//Use this FB if NC-Reference mode is set to "Software Sync" or "Hardware-Sync".
//It is mandatory that the NC encoder parameter "Encoder Sub Mask (absolute range maximum value)" is set to the correct value!
//
//This FB checks the disctance between the falling edge of an reference sensor 
//and the final reference flag of the encoder (e.g. SingleTurn overflow in mode SoftwareSync)
//In case these two signals are very close together, it might be possible that the reference position varied about one motor turn
//depending whether the falling edge of the reference sensor occured before or after the software sync impulse.
//
//The FB reports an OK if the resulting distance if greater or equel than the "MinDistanceInDeg". 
{attribute 'no_check'}
FUNCTION_BLOCK AxSoftSyncDistance EXTENDS FbBase
VAR_OUTPUT CONSTANT
//option settings 
END_VAR
VAR CONSTANT
	DEG_PER_TURN											:	LREAL := 360.0;	
END_VAR
VAR_INPUT
	MinDistanceInDeg										:	LREAL := 45.0; //Minmum required distance between falling edge of sensor and software sync reference impuls (Single turn overflow)   
END_VAR
VAR_IN_OUT
	Axis													:	AXIS_REF;
END_VAR
VAR_OUTPUT
	Distance												: LREAL; //In user units (e.g. mm)
	DistancePerTurn											: LREAL; //In user units (e.g. mm)
	DistanceInDeg											: LREAL; //Resulting distance in degrees	
	OK														: BOOL;  //Inidcates whether the distance between falling edge of sensor and software sync is greater or equal than MinDistanceInDeg  
END_VAR
VAR
(*  Memory *****************************************************)
	LastErrorState											:	INT;
	LastErrorId												:	UDINT;
	ScalingNumerator										:	LREAL;
	ScalingDenumerator										:	LREAL;
	Scaling													:	LREAL;
	RefSystem												:	UDINT;
	RefMode													:	UDINT;
	{attribute 'displaymode':='hex'}
	EncSubMask												:	UDINT;


(*  Timer ******************************************************)

(*  Trigger ****************************************************)

(*  Blocks *****************************************************)
	ReadAdsPara												: ADSREAD := (NetID:= '' , Port:=AMSPORT_R0_NC,TmOut := DEFAULT_ADS_TIMEOUT );

(*  Error ******************************************************)
(*  Dummys *****************************************************)
	{attribute 'hide' := ''}
END_VAR

	(* Check distance between falling edge of reference sensor and deteced sync impulse		*)
	(****************************************************************************************)
	
(* Sequence ********************************************************)
	rtExecute(CLK := Execute);
	CASE state OF
	0 : 
		Busy 												:= FALSE;
		IF NOT Execute THEN
			OK												:= FALSE;
			Done 											:= FALSE;
			Error 											:= FALSE;
			ErrorID 										:= 0;
		END_IF
		IF rtExecute.Q THEN
			ReadAdsPara( Read := FALSE); 
			Busy											:= TRUE;
			Distance										:= 0.0;
			ScalingNumerator								:= 0.0;
			ScalingDenumerator								:= 0.0;
			Scaling											:= 0.0;
			RefSystem										:= 0;
			EncSubMask										:= 0;
			OK												:= FALSE;
			Done 											:= FALSE;
			Error 											:= FALSE;
			ErrorID 										:= 0;
			state 											:= state + 1;
		END_IF
		
		
	(* Read scaling numerator **********************************************)
	1:
		ReadAdsPara(Read:= TRUE,	IDxGrp:=(16#5000+Axis.NcToPlc.AxisId) , IDxOffs:=16#23,LEN:=SIZEOF(ScalingNumerator), DestAddr:=ADR(ScalingNumerator));	
		IF NOT ReadAdsPara.BUSY
		THEN
			IF ReadAdsPara.ERR
			THEN
				Busy										:= FALSE;
				Error										:= TRUE;
				ErrorID										:= ReadAdsPara.ERRID;
				LastErrorState								:= state;
				LastErrorId									:= ErrorId;
				state										:= 0;
			ELSE 
				state										:= state + 1;						
			END_IF
			ReadAdsPara( Read := FALSE);
		END_IF
		
	(* Read scaling denumerator **********************************************)
	2:
		ReadAdsPara(Read:= TRUE,	IDxGrp:=(16#5000+Axis.NcToPlc.AxisId) , IDxOffs:=16#24,LEN:=SIZEOF(ScalingDenumerator), DestAddr:=ADR(ScalingDenumerator));	
		IF NOT ReadAdsPara.BUSY
		THEN
			IF ReadAdsPara.ERR
			THEN
				Busy										:= FALSE;
				Error										:= TRUE;
				ErrorID										:= ReadAdsPara.ERRID;
				LastErrorState									:= state;
				LastErrorId									:= ErrorId;
				state										:= 0;
			ELSE
				Scaling										:= ScalingNumerator / SEL(ScalingDenumerator = 0.0, ScalingDenumerator , 1.0);	
				IF Scaling = 0.0
				THEN
					Busy									:= FALSE;
					Error									:= TRUE;
					ErrorID									:= MC_ERROR_PARAMETER_NOT_CORRECT;
					LastErrorState								:= state;
					LastErrorId									:= ErrorId;
					state									:= 0;	
				ELSE
					state									:= state + 1;
				END_IF					
			END_IF
			ReadAdsPara( Read := FALSE);
		END_IF

	(* Read distance in user units **********************************************)
	3:
		ReadAdsPara(Read:= TRUE,	IDxGrp:=(16#5100+Axis.NcToPlc.AxisId) , IDxOffs:=16#101,LEN:=SIZEOF(Distance), DestAddr:=ADR(Distance));	
		IF NOT ReadAdsPara.BUSY
		THEN
			IF ReadAdsPara.ERR
			THEN
				Busy										:= FALSE;
				Error										:= TRUE;
				ErrorID										:= ReadAdsPara.ERRID;
				LastErrorState									:= state;
				LastErrorId									:= ErrorId;
				state										:= 0;
			ELSE 
				state										:= state + 1;			
			END_IF
			ReadAdsPara( Read := FALSE);
		END_IF
		
	(* Read selected reference system **********************************************)
	4:
		ReadAdsPara(Read:= TRUE,	IDxGrp:=(16#5000+Axis.NcToPlc.AxisId) , IDxOffs:=16#19,LEN:=SIZEOF(RefSystem), DestAddr:=ADR(RefSystem));	
		IF NOT ReadAdsPara.BUSY
		THEN
			IF ReadAdsPara.ERR
			THEN
				Busy										:= FALSE;
				Error										:= TRUE;
				ErrorID										:= ReadAdsPara.ERRID;
				LastErrorState									:= state;
				LastErrorId									:= ErrorId;
				state										:= 0;
			ELSE 
				state										:= state + 1;					
			END_IF
			ReadAdsPara( Read := FALSE);
		END_IF
	
	(* Read selected reference mode **********************************************)
	5:
		ReadAdsPara(Read:= TRUE,	IDxGrp:=(16#5000+Axis.NcToPlc.AxisId) , IDxOffs:=16#107,LEN:=SIZEOF(RefMode), DestAddr:=ADR(RefMode));	
		IF NOT ReadAdsPara.BUSY
		THEN
			IF ReadAdsPara.ERR
			THEN
				Busy										:= FALSE;
				Error										:= TRUE;
				ErrorID										:= ReadAdsPara.ERRID;
				LastErrorState									:= state;
				LastErrorId									:= ErrorId;
				state										:= 0;
			ELSE 
				state										:= state + 1;					
			END_IF
			ReadAdsPara( Read := FALSE);
		END_IF
	
	(* Read EncSubMask (Inc per turn) **********************************************)
	6:
		ReadAdsPara(Read:= TRUE,	IDxGrp:=(16#5000+Axis.NcToPlc.AxisId) , IDxOffs:=16#108,LEN:=SIZEOF(EncSubMask), DestAddr:=ADR(EncSubMask));	
		IF NOT ReadAdsPara.BUSY
		THEN
			IF ReadAdsPara.ERR
			THEN
				Busy										:= FALSE;
				Error										:= TRUE;
				ErrorID										:= ReadAdsPara.ERRID;
				LastErrorState									:= state;
				LastErrorId									:= ErrorId;
				state										:= 0;
			ELSIF EncSubMask = 0
			THEN
				Busy										:= FALSE;
				Error										:= TRUE;
				ErrorID										:= MC_ERROR_PARAMETER_NOT_CORRECT;
				LastErrorState									:= state;
				LastErrorId									:= ErrorId;
				state										:= 0;			
			ELSE
				state										:= state + 1;					
			END_IF
			ReadAdsPara( Read := FALSE);
		END_IF
		
	(* Check reference value ************************************)
	7:
		DistancePerTurn										:= EncSubMask * Scaling;
		DistanceInDeg										:= (DEG_PER_TURN / DistancePerTurn) * Distance;	
																		
		OK													:= ABS(DistanceInDeg) <= DEG_PER_TURN - ABS(MinDistanceInDeg)  
																AND ABS(DistanceInDeg) >= ABS(MinDistanceInDeg) ;							
	
		Busy												:= FALSE;
		Done												:= TRUE;
		state												:= 0;	
	END_CASE

(****************************************************************************************)

END_FUNCTION_BLOCK

(* stored: Version 1.1.0.1, ProductVersion 3.1.4024.3
   POU AxSoftSyncDistance: Id {a88146ba-3783-421b-a8ba-9b0a3a22957d}, SpecialFunc None *)
